(*
SPDX-FileCopyrightText: © 2026 Oleksandr Tiutyk <trofimich@gmail.com>
SPDX-License-Identifier: MIT
License: https://opensource.org/license/mit
*)

INTERFACE IIfElseActivity EXTENDS IExclusiveCompositeActivity

{attribute 'monitoring' := 'call'}
PROPERTY Condition : ICondition
GET
END_GET
SET
END_SET
END_PROPERTY

METHOD Configure
VAR_INPUT
	condition : ICondition; 
	trueActivity : IActivity;
	falseActivity : IActivity;
END_VAR
END_METHOD

{attribute 'monitoring' := 'call'}
PROPERTY FalseActivity : IActivity
GET
END_GET
SET
END_SET
END_PROPERTY

{attribute 'monitoring' := 'call'}
PROPERTY TrueActivity : IActivity
GET
END_GET
SET
END_SET
END_PROPERTY

END_INTERFACE

(* stored: Version 1.1.0.1
   Itf IIfElseActivity: Id {16178d2f-3332-4efd-9137-c92499576b3d}
   Property Condition: Id {6022379b-e762-487a-b202-ef98227acc54}
   Get Get: Id {97ac08d1-4c48-4205-99dc-a466a2da90ff}
   Set Set: Id {0057ab70-c2c0-4b87-a8c1-413e69dff74b}
   Method Configure: Id {c6c70909-4317-4fc7-a63f-e21924dbbf3f}
   Property FalseActivity: Id {68759ad4-444a-491f-804f-0356aa5c7c25}
   Get Get: Id {ca2105be-b58c-48bb-a4b7-c0a379d825b2}
   Set Set: Id {5f7bdd54-5da8-43cf-9d78-4c24945245b0}
   Property TrueActivity: Id {93aee4f4-c6f4-4d2e-926e-53ab0d43d05c}
   Get Get: Id {bafa0510-d2c3-45b0-b482-c7d14c272063}
   Set Set: Id {380346ad-c098-441a-b12c-ac7c0f7b7d5a} *)
